FUNCTION F_VolumeToSteps : REAL
VAR_INPUT
	fVolume 		: REAL; // Volume in µL
    iPumpIndex 		: INT;  // Pump index 1..10
END_VAR
VAR
END_VAR

//Use individual calibration for each pump
F_VolumeToSteps := fVolume / GVL_Settings.aPumpCalibration[iPumpIndex];

END_FUNCTION

(* stored: Version 1.1.0.1, ProductVersion 3.1.4024.12
   POU F_VolumeToSteps: Id {25d1f51c-9d43-4775-9a00-54ad1198621b}, SpecialFunc None *)
